// TIA Portal V18 export
FUNCTION "Enable_machine" : Void   // FC5, LAD
{ S7_Optimized_Access := 'TRUE' }
VERSION : 0.1
// stored: AutoNumber true, IsIECCheckEnabled false, SetENOAutomatically false, UDAEnableTagReadback false
BEGIN

REGION Network 1: Halt Axis
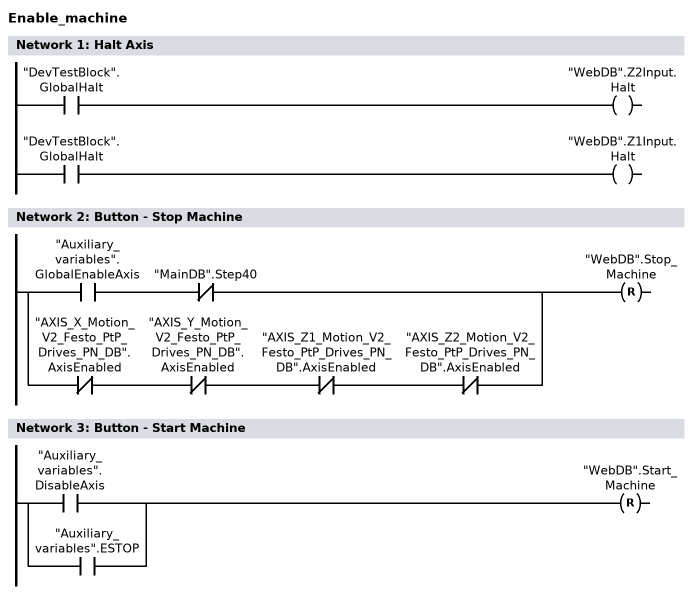
   RUNG wire#powerrail
      Contact( "DevTestBlock".GlobalHalt )
      Coil( "WebDB".Z2Input.Halt )
   END_RUNG
   RUNG wire#powerrail
      Contact( "DevTestBlock".GlobalHalt )
      Coil( "WebDB".Z1Input.Halt )
   END_RUNG
   // the same network as SCL:
   "WebDB".Z2Input.Halt := "DevTestBlock".GlobalHalt;
   "WebDB".Z1Input.Halt := "DevTestBlock".GlobalHalt;
END_REGION

REGION Network 2: Button - Stop Machine
   RUNG wire#powerrail
      Contact( "Auxiliary_variables".GlobalEnableAxis )
      I_Contact( "MainDB".Step40 )
      wire#w1
      R_Coil( "WebDB".Stop_Machine )
   END_RUNG
   RUNG wire#powerrail
      I_Contact( "AXIS_X_Motion_V2_Festo_PtP_Drives_PN_DB".AxisEnabled )
      I_Contact( "AXIS_Y_Motion_V2_Festo_PtP_Drives_PN_DB".AxisEnabled )
      I_Contact( "AXIS_Z1_Motion_V2_Festo_PtP_Drives_PN_DB".AxisEnabled )
      I_Contact( "AXIS_Z2_Motion_V2_Festo_PtP_Drives_PN_DB".AxisEnabled )
   END_RUNG wire#w1
   // the same network as SCL:
   IF ("Auxiliary_variables".GlobalEnableAxis AND NOT "MainDB".Step40) OR (NOT "AXIS_X_Motion_V2_Festo_PtP_Drives_PN_DB".AxisEnabled AND NOT "AXIS_Y_Motion_V2_Festo_PtP_Drives_PN_DB".AxisEnabled AND NOT "AXIS_Z1_Motion_V2_Festo_PtP_Drives_PN_DB".AxisEnabled AND NOT "AXIS_Z2_Motion_V2_Festo_PtP_Drives_PN_DB".AxisEnabled) THEN
       "WebDB".Stop_Machine := FALSE;
   END_IF;
END_REGION

REGION Network 3: Button - Start Machine
   RUNG wire#powerrail
      Contact( "Auxiliary_variables".DisableAxis )
      wire#w1
      R_Coil( "WebDB".Start_Machine )
   END_RUNG
   RUNG wire#powerrail
      Contact( "Auxiliary_variables".ESTOP )
   END_RUNG wire#w1
   // the same network as SCL:
   IF "Auxiliary_variables".DisableAxis OR "Auxiliary_variables".ESTOP THEN
       "WebDB".Start_Machine := FALSE;
   END_IF;
END_REGION
END_FUNCTION
